Yaskawa INFORM job: pointsmerc3TRJ2.JBI

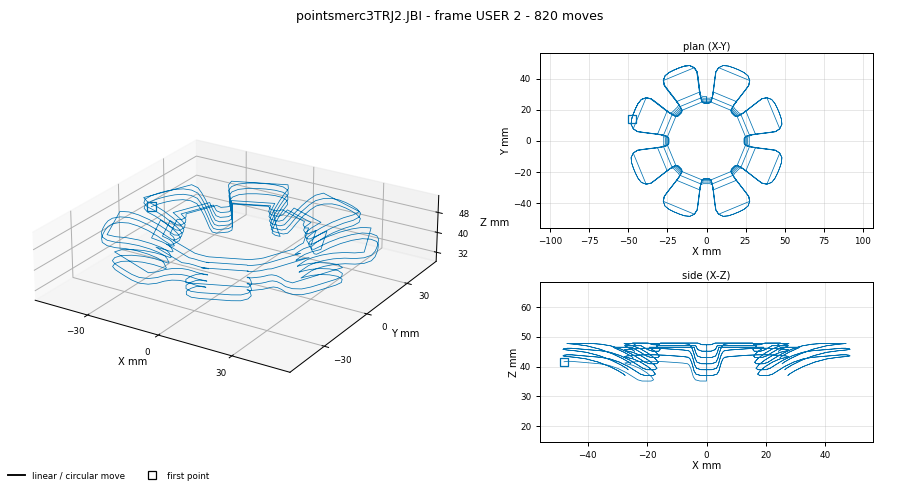
[picture p0: tool path of pointsmerc3TRJ2.JBI in frame USER 2, 820 of 820 moves have a stored position in this frame; points joined in program order, loops and branches not executed]
/JOB
//NAME pointsmerc3TRJ2
//POS
///NPOS 820,0,0,0,0,0
///USER 2
///TOOL 1
///POSTYPE USER
///RECTAN
///RCONF 1,0,0,0,0,0,0,0,0,0,0,0,0,0,0,0,0,0,0,0,0,0,0,0
C00000=-47.960,14.116,41.642,179.9713,-0.0983,0.0000
C00001=-46.852,17.458,41.781,179.9959,-0.0112,0.0000
C00002=-45.474,20.785,41.781,179.9950,-0.0108,0.0000
C00003=-43.894,23.932,41.642,179.9508,-0.0899,0.0000
C00004=-41.848,26.450,41.429,178.7336,-0.9130,0.0000
C00005=-38.982,27.526,41.216,176.7723,-0.3150,0.0000
C00006=-35.890,26.937,40.953,175.4165,2.2977,0.0000
C00007=-32.968,24.818,40.447,175.7483,3.1474,0.0000
C00008=-29.853,22.391,39.399,176.1159,2.8696,0.0000
C00009=-27.005,20.165,37.988,176.7172,2.3719,0.0000
C00010=-24.775,18.500,36.587,178.4223,1.0605,0.0000
C00011=-23.134,17.826,35.561,-161.2162,0.2646,0.0000
C00012=-21.719,18.610,35.152,-154.4517,19.2508,0.0000
C00013=-20.847,19.522,35.134,-156.6171,23.2444,0.0000
C00014=-20.193,20.193,35.146,-155.7569,22.3245,0.0000
C00015=-19.522,20.846,35.134,-154.9222,21.3860,0.0000
C00016=-18.610,21.719,35.152,-158.8420,24.0276,0.0000
C00017=-17.826,23.134,35.561,-179.7208,18.7831,0.0000
C00018=-18.500,24.775,36.587,-178.9391,-1.5774,0.0000
C00019=-20.165,27.005,37.988,-177.6242,-3.2800,0.0000
C00020=-22.391,29.853,39.399,-177.1238,-3.8792,0.0000
C00021=-24.818,32.968,40.447,-176.8439,-4.2453,0.0000
C00022=-26.937,35.890,40.953,-177.6949,-4.5798,0.0000
C00023=-27.526,38.982,41.216,179.6845,-3.2276,0.0000
C00024=-26.450,41.848,41.429,179.0868,-1.2662,0.0000
C00025=-23.932,43.894,41.642,179.9101,-0.0492,0.0000
C00026=-20.785,45.474,41.781,179.9892,-0.0050,0.0000
C00027=-17.458,46.852,41.781,179.9888,-0.0041,0.0000
C00028=-14.116,47.960,41.642,179.9017,-0.0287,0.0000
C00029=-10.888,48.294,41.429,178.4590,0.2497,0.0000
C00030=-8.101,47.028,41.216,177.4938,2.0588,0.0000
C00031=-6.331,44.425,40.953,178.3833,4.8651,0.0000
C00032=-5.763,40.861,40.447,179.2220,5.2308,0.0000
C00033=-5.276,36.942,39.399,179.2849,4.7747,0.0000
C00034=-4.837,33.354,37.988,179.3571,3.9980,0.0000
C00035=-4.437,30.601,36.587,179.6344,1.8654,0.0000
C00036=-3.753,28.963,35.561,-166.2914,-12.9686,0.0000
C00037=-2.199,28.517,35.152,-148.5463,-3.1419,0.0000
C00038=-0.937,28.545,35.134,-147.5179,1.2161,0.0000
C00039=0.000,28.557,35.146,-147.5083,-0.0008,0.0000
C00040=0.000,27.418,37.029,-150.2670,-0.0007,0.0000
C00041=0.833,27.409,37.016,-150.2716,-1.0327,0.0000
C00042=2.024,27.393,37.035,-151.4315,3.4006,0.0000
C00043=3.544,27.900,37.475,-168.9217,11.4487,0.0000
C00044=4.196,29.693,38.576,179.6272,-2.1342,0.0000
C00045=4.590,32.667,40.064,179.4709,-3.5322,0.0000
C00046=5.044,36.489,41.539,179.4511,-3.8692,0.0000
C00047=5.547,40.603,42.621,179.4411,-3.9829,0.0000
C00048=6.113,44.307,43.139,178.8534,-3.5959,0.0000
C00049=7.904,47.004,43.407,178.1982,-1.5163,0.0000
C00050=10.737,48.321,43.623,178.9014,-0.1851,0.0000
C00051=14.024,47.990,43.840,179.9308,0.0202,0.0000
C00052=17.428,46.864,43.981,179.9923,0.0029,0.0000
C00053=20.814,45.461,43.981,179.9925,0.0034,0.0000
C00054=24.018,43.851,43.840,179.9368,0.0347,0.0000
C00055=26.576,41.761,43.623,179.3540,0.9077,0.0000
C00056=27.648,38.826,43.407,179.7985,2.3462,0.0000
C00057=27.007,35.652,43.139,-178.2649,3.3521,0.0000
C00058=24.788,32.633,42.621,-177.5757,3.2100,0.0000
C00059=22.235,29.369,41.539,-177.6492,3.1226,0.0000
C00060=19.854,26.344,40.064,-177.8742,2.8707,0.0000
C00061=18.029,23.963,38.576,-178.7540,1.7725,0.0000
C00062=17.223,22.234,37.475,179.5719,-15.8740,0.0000
C00063=17.939,20.801,37.035,-161.3669,-22.3022,0.0000
C00064=18.793,19.970,37.016,-157.2922,-19.7457,0.0000
C00065=19.387,19.387,37.029,-158.0073,-20.5293,0.0000
C00066=19.970,18.793,37.016,-158.7389,-21.3057,0.0000
C00067=20.801,17.939,37.035,-156.5931,-17.1916,0.0000
C00068=22.234,17.223,37.475,-164.1263,0.4121,0.0000
C00069=23.963,18.029,38.576,178.2271,-1.2454,0.0000
C00070=26.344,19.854,40.064,177.1273,-2.1231,0.0000
C00071=29.369,22.235,41.539,176.8747,-2.3473,0.0000
C00072=32.633,24.788,42.621,176.7872,-2.4205,0.0000
C00073=35.652,27.007,43.139,176.6464,-1.7322,0.0000
C00074=38.826,27.648,43.407,177.6538,0.2014,0.0000
C00075=41.761,26.576,43.623,179.0922,0.6459,0.0000
C00076=43.851,24.018,43.840,179.9653,0.0632,0.0000
C00077=45.461,20.814,43.981,179.9966,0.0075,0.0000
C00078=46.864,17.428,43.981,179.9971,0.0077,0.0000
C00079=47.990,14.024,43.840,179.9798,0.0692,0.0000
C00080=48.321,10.737,43.623,-179.8148,1.0986,0.0000
C00081=47.004,7.904,43.407,-178.4829,1.8012,0.0000
C00082=44.307,6.113,43.139,-176.4033,1.1444,0.0000
C00083=40.603,5.547,42.621,-176.0170,0.5575,0.0000
C00084=36.489,5.044,41.539,-176.1306,0.5476,0.0000
C00085=32.667,4.590,40.064,-176.4677,0.5281,0.0000
C00086=29.693,4.196,38.576,-177.8658,0.3726,0.0000
C00087=27.900,3.544,37.475,168.3398,-10.8552,0.0000
C00088=27.393,2.024,37.035,176.1294,-28.5136,0.0000
C00089=27.409,0.833,37.016,-178.8108,-29.7231,0.0000
C00090=27.418,0.000,37.029,-179.9991,-29.7330,0.0000
C00091=27.409,-0.832,37.016,178.8099,-29.7231,0.0000
C00092=27.393,-2.024,37.035,-176.1268,-28.5126,0.0000
C00093=27.900,-3.544,37.475,-168.3400,-10.8545,0.0000
C00094=29.693,-4.196,38.576,177.8658,0.3726,0.0000
C00095=32.667,-4.590,40.064,176.4677,0.5281,0.0000
C00096=36.489,-5.044,41.539,176.1306,0.5476,0.0000
C00097=40.603,-5.547,42.621,176.0170,0.5575,0.0000
C00098=44.307,-6.113,43.139,176.4033,1.1444,0.0000
C00099=47.004,-7.904,43.407,178.4829,1.8012,0.0000
C00100=48.321,-10.737,43.623,179.8148,1.0986,0.0000
C00101=47.990,-14.024,43.840,-179.9798,0.0692,0.0000
C00102=46.864,-17.428,43.981,-179.9971,0.0077,0.0000
C00103=45.461,-20.814,43.981,-179.9966,0.0075,0.0000
C00104=43.851,-24.018,43.840,-179.9653,0.0632,0.0000
C00105=41.761,-26.576,43.623,-179.0922,0.6459,0.0000
C00106=38.826,-27.648,43.407,-177.6538,0.2014,0.0000
C00107=35.652,-27.007,43.139,-176.6464,-1.7322,0.0000
C00108=32.633,-24.788,42.621,-176.7872,-2.4205,0.0000
C00109=29.369,-22.235,41.539,-176.8747,-2.3473,0.0000
C00110=26.344,-19.854,40.064,-177.1273,-2.1231,0.0000
C00111=23.963,-18.029,38.576,-178.2271,-1.2454,0.0000
C00112=22.234,-17.223,37.475,164.1256,0.4118,0.0000
C00113=20.801,-17.939,37.035,156.5939,-17.1939,0.0000
C00114=19.970,-18.793,37.016,158.7383,-21.3051,0.0000
C00115=19.387,-19.387,37.029,158.0084,-20.5305,0.0000
C00116=18.793,-19.970,37.016,157.2916,-19.7451,0.0000
C00117=17.939,-20.801,37.035,161.3693,-22.3033,0.0000
C00118=17.223,-22.234,37.475,-179.5715,-15.8733,0.0000
C00119=18.029,-23.963,38.576,178.7540,1.7725,0.0000
C00120=19.854,-26.344,40.064,177.8742,2.8707,0.0000
C00121=22.235,-29.369,41.539,177.6492,3.1226,0.0000
C00122=24.788,-32.633,42.621,177.5757,3.2100,0.0000
C00123=27.007,-35.652,43.139,178.2649,3.3521,0.0000
C00124=27.648,-38.826,43.407,-179.7985,2.3462,0.0000
C00125=26.576,-41.761,43.623,-179.3540,0.9077,0.0000
C00126=24.018,-43.851,43.840,-179.9368,0.0347,0.0000
C00127=20.814,-45.461,43.981,-179.9925,0.0034,0.0000
C00128=17.428,-46.864,43.981,-179.9923,0.0029,0.0000
C00129=14.024,-47.990,43.840,-179.9308,0.0202,0.0000
C00130=10.737,-48.321,43.623,-178.9014,-0.1851,0.0000
C00131=7.904,-47.004,43.407,-178.1982,-1.5163,0.0000
C00132=6.113,-44.307,43.139,-178.8534,-3.5959,0.0000
C00133=5.547,-40.603,42.621,-179.4411,-3.9829,0.0000
C00134=5.044,-36.489,41.539,-179.4511,-3.8692,0.0000
C00135=4.590,-32.667,40.064,-179.4709,-3.5322,0.0000
C00136=4.196,-29.693,38.576,-179.6272,-2.1342,0.0000
C00137=3.544,-27.900,37.475,168.9217,11.4487,0.0000
C00138=2.024,-27.393,37.035,151.4315,3.4006,0.0000
C00139=0.833,-27.409,37.016,150.2716,-1.0327,0.0000
C00140=0.000,-27.418,37.029,150.2670,-0.0007,0.0000
C00141=0.000,-27.418,37.029,150.2670,-0.0007,0.0000
C00142=-0.832,-27.409,37.016,150.2716,1.0335,0.0000
C00143=-2.024,-27.393,37.035,151.4324,-3.4028,0.0000
C00144=-3.544,-27.900,37.475,168.9224,-11.4486,0.0000
C00145=-4.196,-29.693,38.576,-179.6272,2.1342,0.0000
C00146=-4.590,-32.667,40.064,-179.4709,3.5322,0.0000
C00147=-5.044,-36.489,41.539,-179.4511,3.8692,0.0000
C00148=-5.547,-40.603,42.621,-179.4411,3.9829,0.0000
C00149=-6.113,-44.307,43.139,-178.8534,3.5959,0.0000
C00150=-7.904,-47.004,43.407,-178.1982,1.5163,0.0000
C00151=-10.737,-48.321,43.623,-178.9014,0.1851,0.0000
C00152=-14.024,-47.990,43.840,-179.9308,-0.0202,0.0000
C00153=-17.428,-46.864,43.981,-179.9923,-0.0029,0.0000
C00154=-20.814,-45.461,43.981,-179.9925,-0.0034,0.0000
C00155=-24.018,-43.851,43.840,-179.9368,-0.0347,0.0000
C00156=-26.576,-41.761,43.623,-179.3540,-0.9077,0.0000
C00157=-27.648,-38.826,43.407,-179.7985,-2.3462,0.0000
C00158=-27.007,-35.652,43.139,178.2649,-3.3521,0.0000
C00159=-24.788,-32.633,42.621,177.5757,-3.2100,0.0000
C00160=-22.235,-29.369,41.539,177.6492,-3.1226,0.0000
C00161=-19.854,-26.344,40.064,177.8742,-2.8707,0.0000
C00162=-18.029,-23.963,38.576,178.7540,-1.7725,0.0000
C00163=-17.223,-22.234,37.475,-179.5719,15.8740,0.0000
C00164=-17.939,-20.801,37.035,161.3669,22.3022,0.0000
C00165=-18.793,-19.970,37.016,157.2922,19.7457,0.0000
C00166=-19.387,-19.387,37.029,158.0073,20.5293,0.0000
C00167=-19.970,-18.793,37.016,158.7389,21.3057,0.0000
C00168=-20.801,-17.939,37.035,156.5931,17.1916,0.0000
C00169=-22.234,-17.223,37.475,164.1263,-0.4121,0.0000
C00170=-23.963,-18.029,38.576,-178.2271,1.2454,0.0000
C00171=-26.344,-19.854,40.064,-177.1273,2.1231,0.0000
C00172=-29.369,-22.235,41.539,-176.8747,2.3473,0.0000
C00173=-32.633,-24.788,42.621,-176.7872,2.4205,0.0000
C00174=-35.652,-27.007,43.139,-176.6464,1.7322,0.0000
C00175=-38.826,-27.648,43.407,-177.6538,-0.2014,0.0000
C00176=-41.761,-26.576,43.623,-179.0922,-0.6459,0.0000
C00177=-43.851,-24.018,43.840,-179.9653,-0.0632,0.0000
C00178=-45.461,-20.814,43.981,-179.9966,-0.0075,0.0000
C00179=-46.864,-17.428,43.981,-179.9971,-0.0077,0.0000
C00180=-47.990,-14.024,43.840,-179.9798,-0.0692,0.0000
C00181=-48.321,-10.737,43.623,179.8148,-1.0986,0.0000
C00182=-47.004,-7.904,43.407,178.4829,-1.8012,0.0000
C00183=-44.307,-6.113,43.139,176.4033,-1.1444,0.0000
C00184=-40.603,-5.547,42.621,176.0170,-0.5575,0.0000
C00185=-36.489,-5.044,41.539,176.1306,-0.5476,0.0000
C00186=-32.667,-4.590,40.064,176.4677,-0.5281,0.0000
C00187=-29.693,-4.196,38.576,177.8658,-0.3726,0.0000
C00188=-27.900,-3.544,37.475,-168.3398,10.8552,0.0000
C00189=-27.393,-2.024,37.035,-176.1294,28.5136,0.0000
C00190=-27.409,-0.833,37.016,178.8108,29.7231,0.0000
C00191=-27.418,0.000,37.029,179.9991,29.7330,0.0000
C00192=-27.409,0.832,37.016,-178.8099,29.7231,0.0000
C00193=-27.393,2.024,37.035,176.1268,28.5126,0.0000
C00194=-27.900,3.544,37.475,168.3400,10.8545,0.0000
C00195=-29.693,4.196,38.576,-177.8658,-0.3726,0.0000
C00196=-32.667,4.590,40.064,-176.4677,-0.5281,0.0000
C00197=-36.489,5.044,41.539,-176.1306,-0.5476,0.0000
C00198=-40.603,5.547,42.621,-176.0170,-0.5575,0.0000
C00199=-44.307,6.113,43.139,-176.4033,-1.1444,0.0000
C00200=-47.004,7.904,43.407,-178.4829,-1.8012,0.0000
C00201=-48.321,10.737,43.623,-179.8148,-1.0986,0.0000
C00202=-47.990,14.024,43.840,179.9798,-0.0692,0.0000
C00203=-46.864,17.428,43.981,179.9971,-0.0077,0.0000
C00204=-45.461,20.814,43.981,179.9966,-0.0075,0.0000
C00205=-43.851,24.018,43.840,179.9653,-0.0632,0.0000
C00206=-41.761,26.576,43.623,179.0922,-0.6459,0.0000
C00207=-38.826,27.648,43.407,177.6538,-0.2014,0.0000
C00208=-35.652,27.007,43.139,176.6464,1.7322,0.0000
C00209=-32.633,24.788,42.621,176.7872,2.4205,0.0000
C00210=-29.369,22.235,41.539,176.8747,2.3473,0.0000
C00211=-26.344,19.854,40.064,177.1273,2.1231,0.0000
C00212=-23.963,18.029,38.576,178.2271,1.2454,0.0000
C00213=-22.234,17.223,37.475,-164.1256,-0.4118,0.0000
C00214=-20.801,17.939,37.035,-156.5939,17.1939,0.0000
C00215=-19.970,18.793,37.016,-158.7383,21.3051,0.0000
C00216=-19.387,19.387,37.029,-158.0084,20.5305,0.0000
C00217=-18.793,19.970,37.016,-157.2916,19.7451,0.0000
C00218=-17.939,20.801,37.035,-161.3693,22.3033,0.0000
C00219=-17.223,22.234,37.475,179.5715,15.8733,0.0000
C00220=-18.029,23.963,38.576,-178.7540,-1.7725,0.0000
C00221=-19.854,26.344,40.064,-177.8742,-2.8707,0.0000
C00222=-22.235,29.369,41.539,-177.6492,-3.1226,0.0000
C00223=-24.788,32.633,42.621,-177.5757,-3.2100,0.0000
C00224=-27.007,35.652,43.139,-178.2649,-3.3521,0.0000
C00225=-27.648,38.826,43.407,179.7985,-2.3462,0.0000
C00226=-26.576,41.761,43.623,179.3540,-0.9077,0.0000
C00227=-24.018,43.851,43.840,179.9368,-0.0347,0.0000
C00228=-20.814,45.461,43.981,179.9925,-0.0034,0.0000
C00229=-17.428,46.864,43.981,179.9923,-0.0029,0.0000
C00230=-14.024,47.990,43.840,179.9308,-0.0202,0.0000
C00231=-10.737,48.321,43.623,178.9014,0.1851,0.0000
C00232=-7.904,47.004,43.407,178.1982,1.5163,0.0000
C00233=-6.113,44.307,43.139,178.8534,3.5959,0.0000
C00234=-5.547,40.603,42.621,179.4411,3.9829,0.0000
C00235=-5.044,36.489,41.539,179.4511,3.8692,0.0000
C00236=-4.590,32.667,40.064,179.4709,3.5322,0.0000
C00237=-4.196,29.693,38.576,179.6272,2.1342,0.0000
C00238=-3.544,27.900,37.475,-168.9224,-11.4486,0.0000
C00239=-2.024,27.393,37.035,-151.4324,-3.4028,0.0000
C00240=-0.832,27.409,37.016,-150.2716,1.0335,0.0000
C00241=0.000,27.418,37.029,-150.2670,-0.0007,0.0000
C00242=0.000,26.383,38.970,-153.7508,-0.0006,0.0000
C00243=0.738,26.377,38.956,-153.7490,-0.8316,0.0000
C00244=1.865,26.371,38.977,-154.9962,3.4534,0.0000
C00245=3.355,26.945,39.448,-171.3719,9.6260,0.0000
C00246=3.987,28.902,40.618,179.6696,-2.0938,0.0000
C00247=4.387,32.102,42.180,179.5989,-2.8366,0.0000
C00248=4.868,36.145,43.705,179.6256,-2.7489,0.0000
C00249=5.395,40.422,44.808,179.6621,-2.5077,0.0000
C00250=5.967,44.227,45.333,179.3497,-2.0954,0.0000
C00251=7.777,46.989,45.603,179.0076,-0.8478,0.0000
C00252=10.643,48.338,45.821,179.4199,-0.1001,0.0000
C00253=13.968,48.009,46.039,179.9653,0.0101,0.0000
C00254=17.410,46.871,46.181,179.9963,0.0014,0.0000
C00255=20.832,45.453,46.181,179.9964,0.0017,0.0000
C00256=24.070,43.824,46.039,179.9683,0.0174,0.0000
C00257=26.655,41.706,45.821,179.6606,0.4809,0.0000
C00258=27.727,38.725,45.603,179.8978,1.3012,0.0000
C00259=27.054,35.493,45.333,-178.9775,1.9413,0.0000
C00260=24.768,32.397,44.808,-178.4649,2.0118,0.0000
C00261=22.116,29.001,43.705,-178.3199,2.2080,0.0000
C00262=19.598,25.801,42.180,-178.2767,2.2889,0.0000
C00263=17.618,23.256,40.618,-178.7526,1.7139,0.0000
C00264=16.680,21.426,39.448,179.1975,-12.8751,0.0000
C00265=17.329,19.966,38.977,-164.2142,-19.9336,0.0000
C00266=18.130,19.173,38.956,-160.1927,-17.6055,0.0000
C00267=18.656,18.656,38.970,-160.7762,-18.2238,0.0000
C00268=19.173,18.130,38.956,-161.3623,-18.8441,0.0000
C00269=19.966,17.329,38.977,-159.3493,-14.8154,0.0000
C00270=21.426,16.680,39.448,-167.1244,0.7826,0.0000
C00271=23.256,17.618,40.618,178.2857,-1.2468,0.0000
C00272=25.801,19.598,42.180,177.7101,-1.7220,0.0000
C00273=29.001,22.116,43.705,177.7910,-1.6789,0.0000
C00274=32.397,24.768,44.808,177.9875,-1.5342,0.0000
C00275=35.493,27.054,45.333,178.0584,-1.0219,0.0000
C00276=38.725,27.727,45.603,178.6988,0.1021,0.0000
C00277=41.706,26.655,45.821,179.5191,0.3394,0.0000
C00278=43.824,24.070,46.039,179.9826,0.0317,0.0000
C00279=45.453,20.832,46.181,179.9983,0.0036,0.0000
C00280=46.871,17.410,46.181,179.9986,0.0037,0.0000
C00281=48.009,13.968,46.039,179.9899,0.0347,0.0000
C00282=48.338,10.643,45.821,-179.8999,0.5801,0.0000
C00283=46.989,7.777,45.603,-179.1520,0.9923,0.0000
C00284=44.227,5.967,45.333,-177.9044,0.6499,0.0000
C00285=40.422,5.395,44.808,-177.4922,0.3376,0.0000
C00286=36.145,4.868,43.705,-177.2510,0.3740,0.0000
C00287=32.102,4.387,42.180,-177.1633,0.4006,0.0000
C00288=28.902,3.987,40.618,-177.9062,0.3302,0.0000
C00289=26.945,3.355,39.448,170.2659,-8.5057,0.0000
C00290=26.371,1.865,38.977,176.1905,-24.9553,0.0000
C00291=26.377,0.738,38.956,-179.0728,-26.2481,0.0000
C00292=26.383,0.000,38.970,-179.9993,-26.2492,0.0000
C00293=26.377,-0.738,38.956,179.0721,-26.2481,0.0000
C00294=26.371,-1.865,38.977,-176.1882,-24.9543,0.0000
C00295=26.945,-3.355,39.448,-170.2662,-8.5050,0.0000
C00296=28.902,-3.987,40.618,177.9062,0.3302,0.0000
C00297=32.102,-4.387,42.180,177.1633,0.4006,0.0000
C00298=36.145,-4.868,43.705,177.2510,0.3740,0.0000
C00299=40.422,-5.395,44.808,177.4922,0.3376,0.0000
C00300=44.227,-5.967,45.333,177.9044,0.6499,0.0000
C00301=46.989,-7.777,45.603,179.1520,0.9923,0.0000
C00302=48.338,-10.643,45.821,179.8999,0.5801,0.0000
C00303=48.009,-13.968,46.039,-179.9899,0.0347,0.0000
C00304=46.871,-17.410,46.181,-179.9986,0.0037,0.0000
C00305=45.453,-20.832,46.181,-179.9983,0.0036,0.0000
C00306=43.824,-24.070,46.039,-179.9826,0.0317,0.0000
C00307=41.706,-26.655,45.821,-179.5191,0.3394,0.0000
C00308=38.725,-27.727,45.603,-178.6988,0.1021,0.0000
C00309=35.493,-27.054,45.333,-178.0584,-1.0219,0.0000
C00310=32.397,-24.768,44.808,-177.9875,-1.5342,0.0000
C00311=29.001,-22.116,43.705,-177.7910,-1.6789,0.0000
C00312=25.801,-19.598,42.180,-177.7101,-1.7220,0.0000
C00313=23.256,-17.618,40.618,-178.2857,-1.2468,0.0000
C00314=21.426,-16.680,39.448,167.1236,0.7823,0.0000
C00315=19.966,-17.329,38.977,159.3500,-14.8176,0.0000
C00316=19.173,-18.130,38.956,161.3618,-18.8436,0.0000
C00317=18.656,-18.656,38.970,160.7770,-18.2247,0.0000
C00318=18.130,-19.173,38.956,160.1923,-17.6051,0.0000
C00319=17.329,-19.966,38.977,164.2165,-19.9345,0.0000
C00320=16.680,-21.426,39.448,-179.1972,-12.8744,0.0000
C00321=17.618,-23.256,40.618,178.7526,1.7139,0.0000
C00322=19.598,-25.801,42.180,178.2767,2.2889,0.0000
C00323=22.116,-29.001,43.705,178.3199,2.2080,0.0000
C00324=24.768,-32.397,44.808,178.4649,2.0118,0.0000
C00325=27.054,-35.493,45.333,178.9775,1.9413,0.0000
C00326=27.727,-38.725,45.603,-179.8978,1.3012,0.0000
C00327=26.655,-41.706,45.821,-179.6606,0.4809,0.0000
C00328=24.070,-43.824,46.039,-179.9683,0.0174,0.0000
C00329=20.832,-45.453,46.181,-179.9964,0.0017,0.0000
C00330=17.410,-46.871,46.181,-179.9963,0.0014,0.0000
C00331=13.968,-48.009,46.039,-179.9653,0.0101,0.0000
C00332=10.643,-48.338,45.821,-179.4199,-0.1001,0.0000
C00333=7.777,-46.989,45.603,-179.0076,-0.8478,0.0000
C00334=5.967,-44.227,45.333,-179.3497,-2.0954,0.0000
C00335=5.395,-40.422,44.808,-179.6621,-2.5077,0.0000
C00336=4.868,-36.145,43.705,-179.6256,-2.7489,0.0000
C00337=4.387,-32.102,42.180,-179.5989,-2.8366,0.0000
C00338=3.987,-28.902,40.618,-179.6696,-2.0938,0.0000
C00339=3.355,-26.945,39.448,171.3719,9.6260,0.0000
C00340=1.865,-26.371,38.977,154.9962,3.4534,0.0000
C00341=0.738,-26.377,38.956,153.7490,-0.8316,0.0000
C00342=0.000,-26.383,38.970,153.7508,-0.0006,0.0000
C00343=0.000,-26.383,38.970,153.7508,-0.0006,0.0000
C00344=-0.738,-26.377,38.956,153.7490,0.8322,0.0000
C00345=-1.865,-26.371,38.977,154.9971,-3.4555,0.0000
C00346=-3.355,-26.945,39.448,171.3727,-9.6258,0.0000
C00347=-3.987,-28.902,40.618,-179.6696,2.0938,0.0000
C00348=-4.387,-32.102,42.180,-179.5989,2.8366,0.0000
C00349=-4.868,-36.145,43.705,-179.6256,2.7489,0.0000
C00350=-5.395,-40.422,44.808,-179.6621,2.5077,0.0000
C00351=-5.967,-44.227,45.333,-179.3497,2.0954,0.0000
C00352=-7.777,-46.989,45.603,-179.0076,0.8478,0.0000
C00353=-10.643,-48.338,45.821,-179.4199,0.1001,0.0000
C00354=-13.968,-48.009,46.039,-179.9653,-0.0101,0.0000
C00355=-17.410,-46.871,46.181,-179.9963,-0.0014,0.0000
C00356=-20.832,-45.453,46.181,-179.9964,-0.0017,0.0000
C00357=-24.070,-43.824,46.039,-179.9683,-0.0174,0.0000
C00358=-26.655,-41.706,45.821,-179.6606,-0.4809,0.0000
C00359=-27.727,-38.725,45.603,-179.8978,-1.3012,0.0000
C00360=-27.054,-35.493,45.333,178.9775,-1.9413,0.0000
C00361=-24.768,-32.397,44.808,178.4649,-2.0118,0.0000
C00362=-22.116,-29.001,43.705,178.3199,-2.2080,0.0000
C00363=-19.598,-25.801,42.180,178.2767,-2.2889,0.0000
C00364=-17.618,-23.256,40.618,178.7526,-1.7139,0.0000
C00365=-16.680,-21.426,39.448,-179.1975,12.8751,0.0000
C00366=-17.329,-19.966,38.977,164.2142,19.9336,0.0000
C00367=-18.130,-19.173,38.956,160.1927,17.6055,0.0000
C00368=-18.656,-18.656,38.970,160.7762,18.2238,0.0000
C00369=-19.173,-18.130,38.956,161.3623,18.8441,0.0000
C00370=-19.966,-17.329,38.977,159.3493,14.8154,0.0000
C00371=-21.426,-16.680,39.448,167.1244,-0.7826,0.0000
C00372=-23.256,-17.618,40.618,-178.2857,1.2468,0.0000
C00373=-25.801,-19.598,42.180,-177.7101,1.7220,0.0000
C00374=-29.001,-22.116,43.705,-177.7910,1.6789,0.0000
C00375=-32.397,-24.768,44.808,-177.9875,1.5342,0.0000
C00376=-35.493,-27.054,45.333,-178.0584,1.0219,0.0000
C00377=-38.725,-27.727,45.603,-178.6988,-0.1021,0.0000
C00378=-41.706,-26.655,45.821,-179.5191,-0.3394,0.0000
C00379=-43.824,-24.070,46.039,-179.9826,-0.0317,0.0000
C00380=-45.453,-20.832,46.181,-179.9983,-0.0036,0.0000
C00381=-46.871,-17.410,46.181,-179.9986,-0.0037,0.0000
C00382=-48.009,-13.968,46.039,-179.9899,-0.0347,0.0000
C00383=-48.338,-10.643,45.821,179.8999,-0.5801,0.0000
C00384=-46.989,-7.777,45.603,179.1520,-0.9923,0.0000
C00385=-44.227,-5.967,45.333,177.9044,-0.6499,0.0000
C00386=-40.422,-5.395,44.808,177.4922,-0.3376,0.0000
C00387=-36.145,-4.868,43.705,177.2510,-0.3740,0.0000
C00388=-32.102,-4.387,42.180,177.1633,-0.4006,0.0000
C00389=-28.902,-3.987,40.618,177.9062,-0.3302,0.0000
C00390=-26.945,-3.355,39.448,-170.2659,8.5057,0.0000
C00391=-26.371,-1.865,38.977,-176.1905,24.9553,0.0000
C00392=-26.377,-0.738,38.956,179.0728,26.2481,0.0000
C00393=-26.383,0.000,38.970,179.9993,26.2492,0.0000
C00394=-26.377,0.738,38.956,-179.0721,26.2481,0.0000
C00395=-26.371,1.865,38.977,176.1882,24.9543,0.0000
C00396=-26.945,3.355,39.448,170.2662,8.5050,0.0000
C00397=-28.902,3.987,40.618,-177.9062,-0.3302,0.0000
C00398=-32.102,4.387,42.180,-177.1633,-0.4006,0.0000
C00399=-36.145,4.868,43.705,-177.2510,-0.3740,0.0000
C00400=-40.422,5.395,44.808,-177.4922,-0.3376,0.0000
C00401=-44.227,5.967,45.333,-177.9044,-0.6499,0.0000
C00402=-46.989,7.777,45.603,-179.1520,-0.9923,0.0000
C00403=-48.338,10.643,45.821,-179.8999,-0.5801,0.0000
C00404=-48.009,13.968,46.039,179.9899,-0.0347,0.0000
C00405=-46.871,17.410,46.181,179.9986,-0.0037,0.0000
C00406=-45.453,20.832,46.181,179.9983,-0.0036,0.0000
C00407=-43.824,24.070,46.039,179.9826,-0.0317,0.0000
C00408=-41.706,26.655,45.821,179.5191,-0.3394,0.0000
C00409=-38.725,27.727,45.603,178.6988,-0.1021,0.0000
C00410=-35.493,27.054,45.333,178.0584,1.0219,0.0000
C00411=-32.397,24.768,44.808,177.9875,1.5342,0.0000
C00412=-29.001,22.116,43.705,177.7910,1.6789,0.0000
C00413=-25.801,19.598,42.180,177.7101,1.7220,0.0000
C00414=-23.256,17.618,40.618,178.2857,1.2468,0.0000
C00415=-21.426,16.680,39.448,-167.1236,-0.7823,0.0000
C00416=-19.966,17.329,38.977,-159.3500,14.8176,0.0000
C00417=-19.173,18.130,38.956,-161.3618,18.8436,0.0000
C00418=-18.656,18.656,38.970,-160.7770,18.2247,0.0000
C00419=-18.130,19.173,38.956,-160.1923,17.6051,0.0000
C00420=-17.329,19.966,38.977,-164.2165,19.9345,0.0000
C00421=-16.680,21.426,39.448,179.1972,12.8744,0.0000
C00422=-17.618,23.256,40.618,-178.7526,-1.7139,0.0000
C00423=-19.598,25.801,42.180,-178.2767,-2.2889,0.0000
C00424=-22.116,29.001,43.705,-178.3199,-2.2080,0.0000
C00425=-24.768,32.397,44.808,-178.4649,-2.0118,0.0000
C00426=-27.054,35.493,45.333,-178.9775,-1.9413,0.0000
C00427=-27.727,38.725,45.603,179.8978,-1.3012,0.0000
C00428=-26.655,41.706,45.821,179.6606,-0.4809,0.0000
C00429=-24.070,43.824,46.039,179.9683,-0.0174,0.0000
C00430=-20.832,45.453,46.181,179.9964,-0.0017,0.0000
C00431=-17.410,46.871,46.181,179.9963,-0.0014,0.0000
C00432=-13.968,48.009,46.039,179.9653,-0.0101,0.0000
C00433=-10.643,48.338,45.821,179.4199,0.1001,0.0000
C00434=-7.777,46.989,45.603,179.0076,0.8478,0.0000
C00435=-5.967,44.227,45.333,179.3497,2.0954,0.0000
C00436=-5.395,40.422,44.808,179.6621,2.5077,0.0000
C00437=-4.868,36.145,43.705,179.6256,2.7489,0.0000
C00438=-4.387,32.102,42.180,179.5989,2.8366,0.0000
C00439=-3.987,28.902,40.618,179.6696,2.0938,0.0000
C00440=-3.355,26.945,39.448,-171.3727,-9.6258,0.0000
C00441=-1.865,26.371,38.977,-154.9971,-3.4555,0.0000
C00442=-0.738,26.377,38.956,-153.7490,0.8322,0.0000
C00443=0.000,26.383,38.970,-153.7508,-0.0006,0.0000
C00444=0.000,25.483,40.978,-158.1137,-0.0004,0.0000
C00445=0.656,25.479,40.963,-158.1034,-0.6202,0.0000
C00446=1.726,25.483,40.985,-159.3485,3.2259,0.0000
C00447=3.194,26.129,41.485,-173.6456,7.5533,0.0000
C00448=3.816,28.261,42.716,179.7442,-1.7639,0.0000
C00449=4.237,31.687,44.335,179.7389,-1.9261,0.0000
C00450=4.757,35.929,45.891,179.8102,-1.4294,0.0000
C00451=5.317,40.329,47.005,179.8913,-0.8234,0.0000
C00452=5.904,44.193,47.531,179.8811,-0.3876,0.0000
C00453=7.727,46.983,47.803,179.9143,-0.0736,0.0000
C00454=27.758,38.686,47.803,179.9915,0.1126,0.0000
C00455=27.074,35.424,47.531,-179.8100,0.3581,0.0000
C00456=24.758,32.277,47.005,-179.4946,0.6591,0.0000
C00457=22.041,28.769,45.891,-179.1233,1.1448,0.0000
C00458=19.410,25.402,44.335,-178.8223,1.5464,0.0000
C00459=17.285,22.682,42.716,-178.9333,1.4280,0.0000
C00460=16.217,20.734,41.485,179.1065,-9.8187,0.0000
C00461=16.798,19.240,40.985,-167.3786,-16.7849,0.0000
C00462=17.553,18.480,40.963,-163.6981,-14.8348,0.0000
C00463=18.019,18.019,40.978,-164.1420,-15.2826,0.0000
C00464=18.480,17.553,40.963,-164.5731,-15.7444,0.0000
C00465=19.240,16.798,40.985,-162.8231,-12.0734,0.0000
C00466=20.735,16.217,41.485,-170.1809,0.8807,0.0000
C00467=22.682,17.285,42.716,178.5717,-1.0663,0.0000
C00468=25.402,19.410,44.335,178.4533,-1.1773,0.0000
C00469=28.769,22.041,45.891,178.8550,-0.8765,0.0000
C00470=32.277,24.758,47.005,179.3409,-0.5054,0.0000
C00471=35.424,27.074,47.531,179.6419,-0.1900,0.0000
C00472=38.686,27.758,47.803,179.8874,0.0085,0.0000
C00473=46.983,7.727,47.803,-179.9264,0.0857,0.0000
C00474=44.193,5.904,47.531,-179.6124,0.1189,0.0000
C00475=40.329,5.317,47.005,-179.1766,0.1086,0.0000
C00476=35.929,4.757,45.891,-178.5706,0.1897,0.0000
C00477=31.687,4.237,44.335,-178.0739,0.2609,0.0000
C00478=28.261,3.816,42.716,-178.2360,0.2557,0.0000
C00479=26.129,3.194,41.485,172.4006,-6.2991,0.0000
C00480=25.483,1.726,40.985,176.5531,-20.6173,0.0000
C00481=25.479,0.656,40.963,-179.3316,-21.8952,0.0000
C00482=25.483,0.000,40.978,-179.9995,-21.8863,0.0000
C00483=25.479,-0.655,40.963,179.3311,-21.8952,0.0000
C00484=25.483,-1.727,40.985,-176.5512,-20.6163,0.0000
C00485=26.129,-3.194,41.485,-172.4009,-6.2984,0.0000
C00486=28.261,-3.816,42.716,178.2360,0.2557,0.0000
C00487=31.687,-4.237,44.335,178.0739,0.2609,0.0000
C00488=35.929,-4.757,45.891,178.5706,0.1897,0.0000
C00489=40.329,-5.317,47.005,179.1766,0.1086,0.0000
C00490=44.193,-5.904,47.531,179.6124,0.1189,0.0000
C00491=46.983,-7.727,47.803,179.9264,0.0857,0.0000
C00492=38.686,-27.758,47.803,-179.8874,0.0085,0.0000
C00493=35.424,-27.074,47.531,-179.6419,-0.1900,0.0000
C00494=32.277,-24.758,47.005,-179.3409,-0.5054,0.0000
C00495=28.769,-22.041,45.891,-178.8550,-0.8765,0.0000
C00496=25.402,-19.410,44.335,-178.4533,-1.1773,0.0000
C00497=22.682,-17.285,42.716,-178.5717,-1.0663,0.0000
C00498=20.734,-16.217,41.485,170.1802,0.8804,0.0000
C00499=19.240,-16.798,40.985,162.8237,-12.0754,0.0000
C00500=18.480,-17.553,40.963,164.5728,-15.7441,0.0000
C00501=18.019,-18.019,40.978,164.1426,-15.2833,0.0000
C00502=17.553,-18.480,40.963,163.6979,-14.8345,0.0000
C00503=16.798,-19.240,40.985,167.3807,-16.7856,0.0000
C00504=16.217,-20.735,41.485,-179.1062,-9.8180,0.0000
C00505=17.285,-22.682,42.716,178.9333,1.4280,0.0000
C00506=19.410,-25.402,44.335,178.8223,1.5464,0.0000
C00507=22.041,-28.769,45.891,179.1233,1.1448,0.0000
C00508=24.758,-32.277,47.005,179.4946,0.6591,0.0000
C00509=27.074,-35.424,47.531,179.8100,0.3581,0.0000
C00510=27.758,-38.686,47.803,-179.9915,0.1126,0.0000
C00511=7.727,-46.983,47.803,-179.9143,-0.0736,0.0000
C00512=5.904,-44.193,47.531,-179.8811,-0.3876,0.0000
C00513=5.317,-40.329,47.005,-179.8913,-0.8234,0.0000
C00514=4.757,-35.929,45.891,-179.8102,-1.4294,0.0000
C00515=4.237,-31.687,44.335,-179.7389,-1.9261,0.0000
C00516=3.816,-28.261,42.716,-179.7442,-1.7639,0.0000
C00517=3.194,-26.129,41.485,173.6456,7.5533,0.0000
C00518=1.726,-25.483,40.985,159.3485,3.2259,0.0000
C00519=0.656,-25.479,40.963,158.1034,-0.6202,0.0000
C00520=0.000,-25.483,40.978,158.1137,-0.0004,0.0000
C00521=0.000,-25.483,40.978,158.1137,-0.0004,0.0000
C00522=-0.655,-25.479,40.963,158.1034,0.6206,0.0000
C00523=-1.727,-25.483,40.985,159.3495,-3.2277,0.0000
C00524=-3.194,-26.129,41.485,173.6463,-7.5530,0.0000
C00525=-3.816,-28.261,42.716,-179.7442,1.7639,0.0000
C00526=-4.237,-31.687,44.335,-179.7389,1.9261,0.0000
C00527=-4.757,-35.929,45.891,-179.8102,1.4294,0.0000
C00528=-5.317,-40.329,47.005,-179.8913,0.8234,0.0000
C00529=-5.904,-44.193,47.531,-179.8811,0.3876,0.0000
C00530=-7.727,-46.983,47.803,-179.9143,0.0736,0.0000
C00531=-27.758,-38.686,47.803,-179.9915,-0.1126,0.0000
C00532=-27.074,-35.424,47.531,179.8100,-0.3581,0.0000
C00533=-24.758,-32.277,47.005,179.4946,-0.6591,0.0000
C00534=-22.041,-28.769,45.891,179.1233,-1.1448,0.0000
C00535=-19.410,-25.402,44.335,178.8223,-1.5464,0.0000
C00536=-17.285,-22.682,42.716,178.9333,-1.4280,0.0000
C00537=-16.217,-20.734,41.485,-179.1065,9.8187,0.0000
C00538=-16.798,-19.240,40.985,167.3786,16.7849,0.0000
C00539=-17.553,-18.480,40.963,163.6981,14.8348,0.0000
C00540=-18.019,-18.019,40.978,164.1420,15.2826,0.0000
C00541=-18.480,-17.553,40.963,164.5731,15.7444,0.0000
C00542=-19.240,-16.798,40.985,162.8231,12.0734,0.0000
C00543=-20.735,-16.217,41.485,170.1809,-0.8807,0.0000
C00544=-22.682,-17.285,42.716,-178.5717,1.0663,0.0000
C00545=-25.402,-19.410,44.335,-178.4533,1.1773,0.0000
C00546=-28.769,-22.041,45.891,-178.8550,0.8765,0.0000
C00547=-32.277,-24.758,47.005,-179.3409,0.5054,0.0000
C00548=-35.424,-27.074,47.531,-179.6419,0.1900,0.0000
C00549=-38.686,-27.758,47.803,-179.8874,-0.0085,0.0000
C00550=-46.983,-7.727,47.803,179.9264,-0.0857,0.0000
C00551=-44.193,-5.904,47.531,179.6124,-0.1189,0.0000
C00552=-40.329,-5.317,47.005,179.1766,-0.1086,0.0000
C00553=-35.929,-4.757,45.891,178.5706,-0.1897,0.0000
C00554=-31.687,-4.237,44.335,178.0739,-0.2609,0.0000
C00555=-28.261,-3.816,42.716,178.2360,-0.2557,0.0000
C00556=-26.129,-3.194,41.485,-172.4006,6.2991,0.0000
C00557=-25.483,-1.726,40.985,-176.5531,20.6173,0.0000
C00558=-25.479,-0.656,40.963,179.3316,21.8952,0.0000
C00559=-25.483,0.000,40.978,179.9995,21.8863,0.0000
C00560=-25.479,0.655,40.963,-179.3311,21.8952,0.0000
C00561=-25.483,1.727,40.985,176.5512,20.6163,0.0000
C00562=-26.129,3.194,41.485,172.4009,6.2984,0.0000
C00563=-28.261,3.816,42.716,-178.2360,-0.2557,0.0000
C00564=-31.687,4.237,44.335,-178.0739,-0.2609,0.0000
C00565=-35.929,4.757,45.891,-178.5706,-0.1897,0.0000
C00566=-40.329,5.317,47.005,-179.1766,-0.1086,0.0000
C00567=-44.193,5.904,47.531,-179.6124,-0.1189,0.0000
C00568=-46.983,7.727,47.803,-179.9264,-0.0857,0.0000
C00569=-38.686,27.758,47.803,179.8874,-0.0085,0.0000
C00570=-35.424,27.074,47.531,179.6419,0.1900,0.0000
C00571=-32.277,24.758,47.005,179.3409,0.5054,0.0000
C00572=-28.769,22.041,45.891,178.8550,0.8765,0.0000
C00573=-25.402,19.410,44.335,178.4533,1.1773,0.0000
C00574=-22.682,17.285,42.716,178.5717,1.0663,0.0000
C00575=-20.734,16.217,41.485,-170.1802,-0.8804,0.0000
C00576=-19.240,16.798,40.985,-162.8237,12.0754,0.0000
C00577=-18.480,17.553,40.963,-164.5728,15.7441,0.0000
C00578=-18.019,18.019,40.978,-164.1426,15.2833,0.0000
C00579=-17.553,18.480,40.963,-163.6979,14.8345,0.0000
C00580=-16.798,19.240,40.985,-167.3807,16.7856,0.0000
C00581=-16.217,20.735,41.485,179.1062,9.8180,0.0000
C00582=-17.285,22.682,42.716,-178.9333,-1.4280,0.0000
C00583=-19.410,25.402,44.335,-178.8223,-1.5464,0.0000
C00584=-22.041,28.769,45.891,-179.1233,-1.1448,0.0000
C00585=-24.758,32.277,47.005,-179.4946,-0.6591,0.0000
C00586=-27.074,35.424,47.531,-179.8100,-0.3581,0.0000
C00587=-27.758,38.686,47.803,179.9915,-0.1126,0.0000
C00588=-7.727,46.983,47.803,179.9143,0.0736,0.0000
C00589=-5.904,44.193,47.531,179.8811,0.3876,0.0000
C00590=-5.317,40.329,47.005,179.8913,0.8234,0.0000
C00591=-4.757,35.929,45.891,179.8102,1.4294,0.0000
C00592=-4.237,31.687,44.335,179.7389,1.9261,0.0000
C00593=-3.816,28.261,42.716,179.7442,1.7639,0.0000
C00594=-3.194,26.129,41.485,-173.6463,-7.5530,0.0000
C00595=-1.727,25.483,40.985,-159.3495,-3.2277,0.0000
C00596=-0.655,25.479,40.963,-158.1034,0.6206,0.0000
C00597=0.000,25.483,40.978,-158.1137,-0.0004,0.0000
C00598=0.000,24.757,43.054,-163.5138,-0.0002,0.0000
C00599=0.589,24.754,43.039,-163.4920,-0.4122,0.0000
C00600=1.615,24.766,43.062,-164.5921,2.6504,0.0000
C00601=3.068,25.489,43.586,-175.7793,5.2659,0.0000
C00602=3.695,27.804,44.865,179.8395,-1.1765,0.0000
C00603=4.151,31.448,46.521,179.8907,-0.8261,0.0000
C00604=19.301,25.172,46.521,-179.4931,0.6614,0.0000
C00605=17.048,22.273,44.865,-179.2815,0.9454,0.0000
C00606=15.854,20.193,43.586,179.2457,-6.7028,0.0000
C00607=16.370,18.654,43.062,-170.8582,-12.7306,0.0000
C00608=17.087,17.920,43.039,-167.8734,-11.2933,0.0000
C00609=17.506,17.506,43.054,-168.1802,-11.5757,0.0000
C00610=17.920,17.087,43.039,-168.4559,-11.8884,0.0000
C00611=18.654,16.370,43.062,-167.1106,-8.9135,0.0000
C00612=20.193,15.854,43.586,-173.2972,0.7493,0.0000
C00613=22.273,17.048,44.865,179.0546,-0.7184,0.0000
C00614=25.172,19.301,46.521,179.3386,-0.5068,0.0000
C00615=31.448,4.151,46.521,-179.1739,0.1093,0.0000
C00616=27.804,3.695,44.865,-178.8235,0.1604,0.0000
C00617=25.489,3.068,43.586,174.7199,-4.2029,0.0000
C00618=24.766,1.615,43.062,177.2510,-15.3911,0.0000
C00619=24.754,0.589,43.039,-179.5701,-16.5075,0.0000
C00620=24.757,0.000,43.054,-179.9998,-16.4862,0.0000
C00621=24.754,-0.589,43.039,179.5700,-16.5075,0.0000
C00622=24.766,-1.615,43.062,-177.2494,-15.3902,0.0000
C00623=25.489,-3.068,43.586,-174.7201,-4.2024,0.0000
C00624=27.804,-3.695,44.865,178.8235,0.1604,0.0000
C00625=31.448,-4.151,46.521,179.1739,0.1093,0.0000
C00626=25.172,-19.301,46.521,-179.3386,-0.5068,0.0000
C00627=22.273,-17.048,44.865,-179.0546,-0.7184,0.0000
C00628=20.193,-15.854,43.586,173.2966,0.7491,0.0000
C00629=18.654,-16.370,43.062,167.1110,-8.9152,0.0000
C00630=17.920,-17.087,43.039,168.4558,-11.8883,0.0000
C00631=17.506,-17.506,43.054,168.1805,-11.5761,0.0000
C00632=17.087,-17.920,43.039,167.8733,-11.2932,0.0000
C00633=16.370,-18.654,43.062,170.8599,-12.7311,0.0000
C00634=15.854,-20.193,43.586,-179.2456,-6.7022,0.0000
C00635=17.048,-22.273,44.865,179.2815,0.9454,0.0000
C00636=19.301,-25.172,46.521,179.4931,0.6614,0.0000
C00637=4.151,-31.448,46.521,-179.8907,-0.8261,0.0000
C00638=3.695,-27.804,44.865,-179.8395,-1.1765,0.0000
C00639=3.068,-25.489,43.586,175.7793,5.2659,0.0000
C00640=1.615,-24.766,43.062,164.5921,2.6504,0.0000
C00641=0.589,-24.754,43.039,163.4920,-0.4122,0.0000
C00642=0.000,-24.757,43.054,163.5138,-0.0002,0.0000
C00643=0.000,-24.757,43.054,163.5138,-0.0002,0.0000
C00644=-0.589,-24.754,43.039,163.4920,0.4123,0.0000
C00645=-1.615,-24.766,43.062,164.5929,-2.6519,0.0000
C00646=-3.068,-25.489,43.586,175.7798,-5.2656,0.0000
C00647=-3.695,-27.804,44.865,-179.8395,1.1765,0.0000
C00648=-4.151,-31.448,46.521,-179.8907,0.8261,0.0000
C00649=-19.301,-25.172,46.521,179.4931,-0.6614,0.0000
C00650=-17.048,-22.273,44.865,179.2815,-0.9454,0.0000
C00651=-15.854,-20.193,43.586,-179.2457,6.7028,0.0000
C00652=-16.370,-18.654,43.062,170.8582,12.7306,0.0000
C00653=-17.087,-17.920,43.039,167.8734,11.2933,0.0000
C00654=-17.506,-17.506,43.054,168.1802,11.5757,0.0000
C00655=-17.920,-17.087,43.039,168.4559,11.8884,0.0000
C00656=-18.654,-16.370,43.062,167.1106,8.9135,0.0000
C00657=-20.193,-15.854,43.586,173.2972,-0.7493,0.0000
C00658=-22.273,-17.048,44.865,-179.0546,0.7184,0.0000
C00659=-25.172,-19.301,46.521,-179.3386,0.5068,0.0000
C00660=-31.448,-4.151,46.521,179.1739,-0.1093,0.0000
C00661=-27.804,-3.695,44.865,178.8235,-0.1604,0.0000
C00662=-25.489,-3.068,43.586,-174.7199,4.2029,0.0000
C00663=-24.766,-1.615,43.062,-177.2510,15.3911,0.0000
C00664=-24.754,-0.589,43.039,179.5701,16.5075,0.0000
C00665=-24.757,0.000,43.054,179.9998,16.4862,0.0000
C00666=-24.754,0.589,43.039,-179.5700,16.5075,0.0000
C00667=-24.766,1.615,43.062,177.2494,15.3902,0.0000
C00668=-25.489,3.068,43.586,174.7201,4.2024,0.0000
C00669=-27.804,3.695,44.865,-178.8235,-0.1604,0.0000
C00670=-31.448,4.151,46.521,-179.1739,-0.1093,0.0000
C00671=-25.172,19.301,46.521,179.3386,0.5068,0.0000
C00672=-22.273,17.048,44.865,179.0546,0.7184,0.0000
C00673=-20.193,15.854,43.586,-173.2966,-0.7491,0.0000
C00674=-18.654,16.370,43.062,-167.1110,8.9152,0.0000
C00675=-17.920,17.087,43.039,-168.4558,11.8883,0.0000
C00676=-17.506,17.506,43.054,-168.1805,11.5761,0.0000
C00677=-17.087,17.920,43.039,-167.8733,11.2932,0.0000
C00678=-16.370,18.654,43.062,-170.8599,12.7311,0.0000
C00679=-15.854,20.193,43.586,179.2456,6.7022,0.0000
C00680=-17.048,22.273,44.865,-179.2815,-0.9454,0.0000
C00681=-19.301,25.172,46.521,-179.4931,-0.6614,0.0000
C00682=-4.151,31.448,46.521,179.8907,0.8261,0.0000
C00683=-3.695,27.804,44.865,179.8395,1.1765,0.0000
C00684=-3.068,25.489,43.586,-175.7798,-5.2656,0.0000
C00685=-1.615,24.766,43.062,-164.5929,-2.6519,0.0000
C00686=-0.589,24.754,43.039,-163.4920,0.4123,0.0000
C00687=0.000,24.757,43.054,-163.5138,-0.0002,0.0000
C00688=0.000,24.250,45.195,-170.0572,-0.0001,0.0000
C00689=0.543,24.247,45.179,-170.0200,-0.2212,0.0000
C00690=1.537,24.267,45.203,-170.7882,1.6931,0.0000
C00691=2.986,25.071,45.744,-177.8426,2.7768,0.0000
C00692=3.633,27.569,47.051,179.9492,-0.3847,0.0000
C00693=16.925,22.063,47.051,-179.7639,0.3080,0.0000
C00694=15.616,19.839,45.744,179.5599,-3.4882,0.0000
C00695=16.072,18.246,45.203,-174.6583,-7.7031,0.0000
C00696=16.761,17.529,45.179,-172.7509,-6.8814,0.0000
C00697=17.148,17.148,45.195,-172.9339,-7.0129,0.0000
C00698=17.529,16.762,45.179,-173.0637,-7.1966,0.0000
C00699=18.246,16.072,45.203,-172.2635,-5.2923,0.0000
C00700=19.839,15.616,45.744,-176.5120,0.4394,0.0000
C00701=22.063,16.925,47.051,179.6920,-0.2361,0.0000
C00702=27.569,3.633,47.051,-179.6153,0.0508,0.0000
C00703=25.071,2.986,45.744,177.2213,-2.1549,0.0000
C00704=24.267,1.537,45.203,178.2848,-9.2077,0.0000
C00705=24.247,0.543,45.179,-179.7754,-9.9800,0.0000
C00706=24.250,0.000,45.195,-179.9999,-9.9428,0.0000
C00707=24.247,-0.542,45.179,179.7755,-9.9800,0.0000
C00708=24.267,-1.537,45.203,-178.2839,-9.2071,0.0000
C00709=25.071,-2.986,45.744,-177.2215,-2.1546,0.0000
C00710=27.569,-3.633,47.051,179.6153,0.0508,0.0000
C00711=22.063,-16.925,47.051,-179.6920,-0.2361,0.0000
C00712=19.839,-15.616,45.744,176.5117,0.4393,0.0000
C00713=18.246,-16.072,45.203,172.2637,-5.2934,0.0000
C00714=17.529,-16.761,45.179,173.0637,-7.1966,0.0000
C00715=17.148,-17.148,45.195,172.9340,-7.0129,0.0000
C00716=16.762,-17.529,45.179,172.7509,-6.8814,0.0000
C00717=16.072,-18.246,45.203,174.6594,-7.7033,0.0000
C00718=15.616,-19.839,45.744,-179.5598,-3.4879,0.0000
C00719=16.925,-22.063,47.051,179.7639,0.3080,0.0000
C00720=3.633,-27.569,47.051,-179.9492,-0.3847,0.0000
C00721=2.986,-25.071,45.744,177.8426,2.7768,0.0000
C00722=1.537,-24.267,45.203,170.7882,1.6931,0.0000
C00723=0.543,-24.247,45.179,170.0200,-0.2212,0.0000
C00724=0.000,-24.250,45.195,170.0572,-0.0001,0.0000
C00725=0.000,-24.250,45.195,170.0572,-0.0001,0.0000
C00726=-0.542,-24.247,45.179,170.0200,0.2211,0.0000
C00727=-1.537,-24.267,45.203,170.7888,-1.6940,0.0000
C00728=-2.986,-25.071,45.744,177.8429,-2.7766,0.0000
C00729=-3.633,-27.569,47.051,-179.9492,0.3847,0.0000
C00730=-16.925,-22.063,47.051,179.7639,-0.3080,0.0000
C00731=-15.616,-19.839,45.744,-179.5599,3.4882,0.0000
C00732=-16.072,-18.246,45.203,174.6583,7.7031,0.0000
C00733=-16.761,-17.529,45.179,172.7509,6.8814,0.0000
C00734=-17.148,-17.148,45.195,172.9339,7.0129,0.0000
C00735=-17.529,-16.762,45.179,173.0637,7.1966,0.0000
C00736=-18.246,-16.072,45.203,172.2635,5.2923,0.0000
C00737=-19.839,-15.616,45.744,176.5120,-0.4394,0.0000
C00738=-22.063,-16.925,47.051,-179.6920,0.2361,0.0000
C00739=-27.569,-3.633,47.051,179.6153,-0.0508,0.0000
C00740=-25.071,-2.986,45.744,-177.2213,2.1549,0.0000
C00741=-24.267,-1.537,45.203,-178.2848,9.2077,0.0000
C00742=-24.247,-0.543,45.179,179.7754,9.9800,0.0000
C00743=-24.250,0.000,45.195,179.9999,9.9428,0.0000
C00744=-24.247,0.542,45.179,-179.7755,9.9800,0.0000
C00745=-24.267,1.537,45.203,178.2839,9.2071,0.0000
C00746=-25.071,2.986,45.744,177.2215,2.1546,0.0000
C00747=-27.569,3.633,47.051,-179.6153,-0.0508,0.0000
C00748=-22.063,16.925,47.051,179.6920,0.2361,0.0000
C00749=-19.839,15.616,45.744,-176.5117,-0.4393,0.0000
C00750=-18.246,16.072,45.203,-172.2637,5.2934,0.0000
C00751=-17.529,16.761,45.179,-173.0637,7.1966,0.0000
C00752=-17.148,17.148,45.195,-172.9340,7.0129,0.0000
C00753=-16.762,17.529,45.179,-172.7509,6.8814,0.0000
C00754=-16.072,18.246,45.203,-174.6594,7.7033,0.0000
C00755=-15.616,19.839,45.744,179.5598,3.4879,0.0000
C00756=-16.925,22.063,47.051,-179.7639,-0.3080,0.0000
C00757=-3.633,27.569,47.051,179.9492,0.3847,0.0000
C00758=-2.986,25.071,45.744,-177.8429,-2.7766,0.0000
C00759=-1.537,24.267,45.203,-170.7888,-1.6940,0.0000
C00760=-0.542,24.247,45.179,-170.0200,0.2211,0.0000
C00761=0.000,24.250,45.195,-170.0572,-0.0001,0.0000
C00762=0.000,24.012,47.382,-177.6951,-0.0000,0.0000
C00763=0.521,24.008,47.366,-177.6395,-0.0488,0.0000
C00764=1.501,24.033,47.390,-177.8943,0.3992,0.0000
C00765=2.955,24.917,47.939,-179.9400,0.0782,0.0000
C00766=15.529,19.709,47.939,179.9872,-0.0977,0.0000
C00767=15.933,18.055,47.390,-178.7930,-1.7711,0.0000
C00768=16.608,17.344,47.366,-178.2959,-1.6344,0.0000
C00769=16.979,16.979,47.382,-178.3698,-1.6296,0.0000
C00770=17.344,16.608,47.366,-178.3649,-1.7034,0.0000
C00771=18.055,15.933,47.390,-178.2286,-1.2060,0.0000
C00772=19.709,15.529,47.939,-179.9024,0.0128,0.0000
C00773=24.917,2.955,47.939,179.9218,-0.0600,0.0000
C00774=24.033,1.501,47.390,179.6005,-2.1056,0.0000
C00775=24.008,0.521,47.366,-179.9512,-2.3605,0.0000
C00776=24.012,0.000,47.382,-180.0000,-2.3049,0.0000
C00777=24.008,-0.521,47.366,179.9512,-2.3605,0.0000
C00778=24.033,-1.501,47.390,-179.6004,-2.1053,0.0000
C00779=24.917,-2.955,47.939,-179.9219,-0.0600,0.0000
C00780=19.709,-15.529,47.939,179.9023,0.0128,0.0000
C00781=18.055,-15.933,47.390,178.2285,-1.2064,0.0000
C00782=17.344,-16.608,47.366,178.3649,-1.7034,0.0000
C00783=16.979,-16.979,47.382,178.3698,-1.6296,0.0000
C00784=16.608,-17.344,47.366,178.2959,-1.6344,0.0000
C00785=15.933,-18.055,47.390,178.7934,-1.7710,0.0000
C00786=15.529,-19.709,47.939,-179.9872,-0.0976,0.0000
C00787=2.955,-24.917,47.939,179.9400,0.0782,0.0000
C00788=1.501,-24.033,47.390,177.8943,0.3992,0.0000
C00789=0.521,-24.008,47.366,177.6395,-0.0488,0.0000
C00790=0.000,-24.012,47.382,177.6951,-0.0000,0.0000
C00791=0.000,-24.012,47.382,177.6951,-0.0000,0.0000
C00792=-0.521,-24.008,47.366,177.6395,0.0488,0.0000
C00793=-1.501,-24.033,47.390,177.8946,-0.3994,0.0000
C00794=-2.955,-24.917,47.939,179.9400,-0.0781,0.0000
C00795=-15.529,-19.709,47.939,-179.9872,0.0977,0.0000
C00796=-15.933,-18.055,47.390,178.7930,1.7711,0.0000
C00797=-16.608,-17.344,47.366,178.2959,1.6344,0.0000
C00798=-16.979,-16.979,47.382,178.3698,1.6296,0.0000
C00799=-17.344,-16.608,47.366,178.3649,1.7034,0.0000
C00800=-18.055,-15.933,47.390,178.2286,1.2060,0.0000
C00801=-19.709,-15.529,47.939,179.9024,-0.0128,0.0000
C00802=-24.917,-2.955,47.939,-179.9218,0.0600,0.0000
C00803=-24.033,-1.501,47.390,-179.6005,2.1056,0.0000
C00804=-24.008,-0.521,47.366,179.9512,2.3605,0.0000
C00805=-24.012,0.000,47.382,180.0000,2.3049,0.0000
C00806=-24.008,0.521,47.366,-179.9512,2.3605,0.0000
C00807=-24.033,1.501,47.390,179.6004,2.1053,0.0000
C00808=-24.917,2.955,47.939,179.9219,0.0600,0.0000
C00809=-19.709,15.529,47.939,-179.9023,-0.0128,0.0000
C00810=-18.055,15.933,47.390,-178.2285,1.2064,0.0000
C00811=-17.344,16.608,47.366,-178.3649,1.7034,0.0000
C00812=-16.979,16.979,47.382,-178.3698,1.6296,0.0000
C00813=-16.608,17.344,47.366,-178.2959,1.6344,0.0000
C00814=-15.933,18.055,47.390,-178.7934,1.7710,0.0000
C00815=-15.529,19.709,47.939,179.9872,0.0976,0.0000
C00816=-2.955,24.917,47.939,-179.9400,-0.0781,0.0000
C00817=-1.501,24.033,47.390,-177.8946,-0.3994,0.0000
C00818=-0.521,24.008,47.366,-177.6395,0.0488,0.0000
C00819=0.000,24.012,47.382,-177.6951,-0.0000,0.0000
//INST
///DATE 2021/02/10 13:51
///COMM
///ATTR SC,RW,RJ
////FRAME USER 2
///GROUP1 RB1
NOP
MOVL C00000
MOVL C00001
MOVL C00002
MOVL C00003
MOVL C00004
MOVL C00005
MOVL C00006
MOVL C00007
MOVL C00008
MOVL C00009
MOVL C00010
MOVL C00011
MOVL C00012
MOVL C00013
MOVL C00014
MOVL C00015
MOVL C00016
MOVL C00017
MOVL C00018
MOVL C00019
MOVL C00020
MOVL C00021
MOVL C00022
MOVL C00023
MOVL C00024
MOVL C00025
MOVL C00026
MOVL C00027
MOVL C00028
MOVL C00029
MOVL C00030
MOVL C00031
MOVL C00032
MOVL C00033
MOVL C00034
MOVL C00035
MOVL C00036
MOVL C00037
MOVL C00038
MOVL C00039
MOVL C00040
MOVL C00041
MOVL C00042
MOVL C00043
MOVL C00044
MOVL C00045
MOVL C00046
MOVL C00047
MOVL C00048
MOVL C00049
MOVL C00050
MOVL C00051
MOVL C00052
MOVL C00053
MOVL C00054
MOVL C00055
MOVL C00056
MOVL C00057
MOVL C00058
MOVL C00059
MOVL C00060
MOVL C00061
MOVL C00062
MOVL C00063
MOVL C00064
MOVL C00065
MOVL C00066
MOVL C00067
MOVL C00068
MOVL C00069
MOVL C00070
MOVL C00071
MOVL C00072
MOVL C00073
MOVL C00074
MOVL C00075
MOVL C00076
MOVL C00077
MOVL C00078
MOVL C00079
MOVL C00080
MOVL C00081
MOVL C00082
MOVL C00083
MOVL C00084
MOVL C00085
MOVL C00086
MOVL C00087
MOVL C00088
MOVL C00089
MOVL C00090
MOVL C00091
MOVL C00092
MOVL C00093
MOVL C00094
MOVL C00095
MOVL C00096
MOVL C00097
MOVL C00098
MOVL C00099
MOVL C00100
MOVL C00101
MOVL C00102
MOVL C00103
MOVL C00104
MOVL C00105
MOVL C00106
MOVL C00107
MOVL C00108
MOVL C00109
MOVL C00110
MOVL C00111
MOVL C00112
MOVL C00113
MOVL C00114
MOVL C00115
MOVL C00116
MOVL C00117
MOVL C00118
MOVL C00119
MOVL C00120
MOVL C00121
MOVL C00122
MOVL C00123
MOVL C00124
MOVL C00125
MOVL C00126
MOVL C00127
MOVL C00128
MOVL C00129
MOVL C00130
MOVL C00131
MOVL C00132
MOVL C00133
MOVL C00134
MOVL C00135
MOVL C00136
MOVL C00137
MOVL C00138
MOVL C00139
MOVL C00140
MOVL C00141
MOVL C00142
MOVL C00143
MOVL C00144
MOVL C00145
MOVL C00146
MOVL C00147
MOVL C00148
MOVL C00149
MOVL C00150
MOVL C00151
MOVL C00152
MOVL C00153
MOVL C00154
MOVL C00155
MOVL C00156
MOVL C00157
MOVL C00158
MOVL C00159
MOVL C00160
MOVL C00161
MOVL C00162
MOVL C00163
MOVL C00164
MOVL C00165
MOVL C00166
MOVL C00167
MOVL C00168
MOVL C00169
MOVL C00170
MOVL C00171
MOVL C00172
MOVL C00173
MOVL C00174
MOVL C00175
MOVL C00176
MOVL C00177
MOVL C00178
MOVL C00179
MOVL C00180
MOVL C00181
MOVL C00182
MOVL C00183
MOVL C00184
MOVL C00185
MOVL C00186
MOVL C00187
MOVL C00188
MOVL C00189
MOVL C00190
MOVL C00191
MOVL C00192
MOVL C00193
MOVL C00194
MOVL C00195
MOVL C00196
MOVL C00197
MOVL C00198
MOVL C00199
MOVL C00200
MOVL C00201
MOVL C00202
MOVL C00203
MOVL C00204
MOVL C00205
MOVL C00206
MOVL C00207
MOVL C00208
MOVL C00209
MOVL C00210
MOVL C00211
MOVL C00212
MOVL C00213
MOVL C00214
MOVL C00215
MOVL C00216
MOVL C00217
MOVL C00218
MOVL C00219
MOVL C00220
MOVL C00221
MOVL C00222
MOVL C00223
MOVL C00224
MOVL C00225
MOVL C00226
MOVL C00227
MOVL C00228
MOVL C00229
MOVL C00230
MOVL C00231
MOVL C00232
MOVL C00233
MOVL C00234
MOVL C00235
MOVL C00236
MOVL C00237
MOVL C00238
MOVL C00239
MOVL C00240
MOVL C00241
MOVL C00242
MOVL C00243
MOVL C00244
MOVL C00245
MOVL C00246
MOVL C00247
MOVL C00248
MOVL C00249
MOVL C00250
MOVL C00251
MOVL C00252
MOVL C00253
MOVL C00254
MOVL C00255
MOVL C00256
MOVL C00257
MOVL C00258
MOVL C00259
MOVL C00260
MOVL C00261
MOVL C00262
MOVL C00263
MOVL C00264
MOVL C00265
MOVL C00266
MOVL C00267
MOVL C00268
MOVL C00269
MOVL C00270
MOVL C00271
MOVL C00272
MOVL C00273
MOVL C00274
MOVL C00275
MOVL C00276
MOVL C00277
MOVL C00278
MOVL C00279
MOVL C00280
MOVL C00281
MOVL C00282
MOVL C00283
MOVL C00284
MOVL C00285
MOVL C00286
MOVL C00287
MOVL C00288
MOVL C00289
MOVL C00290
MOVL C00291
MOVL C00292
MOVL C00293
MOVL C00294
MOVL C00295
MOVL C00296
MOVL C00297
MOVL C00298
MOVL C00299
MOVL C00300
MOVL C00301
MOVL C00302
MOVL C00303
MOVL C00304
MOVL C00305
MOVL C00306
MOVL C00307
MOVL C00308
MOVL C00309
MOVL C00310
MOVL C00311
MOVL C00312
MOVL C00313
MOVL C00314
MOVL C00315
MOVL C00316
MOVL C00317
MOVL C00318
MOVL C00319
MOVL C00320
MOVL C00321
MOVL C00322
MOVL C00323
MOVL C00324
MOVL C00325
MOVL C00326
MOVL C00327
MOVL C00328
MOVL C00329
MOVL C00330
MOVL C00331
MOVL C00332
MOVL C00333
MOVL C00334
MOVL C00335
MOVL C00336
MOVL C00337
MOVL C00338
MOVL C00339
MOVL C00340
MOVL C00341
MOVL C00342
MOVL C00343
MOVL C00344
MOVL C00345
MOVL C00346
MOVL C00347
MOVL C00348
MOVL C00349
MOVL C00350
MOVL C00351
MOVL C00352
MOVL C00353
MOVL C00354
MOVL C00355
MOVL C00356
MOVL C00357
MOVL C00358
MOVL C00359
MOVL C00360
MOVL C00361
MOVL C00362
MOVL C00363
MOVL C00364
MOVL C00365
MOVL C00366
MOVL C00367
MOVL C00368
MOVL C00369
MOVL C00370
MOVL C00371
MOVL C00372
MOVL C00373
MOVL C00374
MOVL C00375
MOVL C00376
MOVL C00377
MOVL C00378
MOVL C00379
MOVL C00380
MOVL C00381
MOVL C00382
MOVL C00383
MOVL C00384
MOVL C00385
MOVL C00386
MOVL C00387
MOVL C00388
MOVL C00389
MOVL C00390
MOVL C00391
MOVL C00392
MOVL C00393
MOVL C00394
MOVL C00395
MOVL C00396
MOVL C00397
MOVL C00398
MOVL C00399
MOVL C00400
MOVL C00401
MOVL C00402
MOVL C00403
MOVL C00404
MOVL C00405
MOVL C00406
MOVL C00407
MOVL C00408
MOVL C00409
MOVL C00410
MOVL C00411
MOVL C00412
MOVL C00413
MOVL C00414
MOVL C00415
MOVL C00416
MOVL C00417
MOVL C00418
MOVL C00419
MOVL C00420
MOVL C00421
MOVL C00422
MOVL C00423
MOVL C00424
MOVL C00425
MOVL C00426
MOVL C00427
MOVL C00428
MOVL C00429
MOVL C00430
MOVL C00431
MOVL C00432
MOVL C00433
MOVL C00434
MOVL C00435
MOVL C00436
MOVL C00437
MOVL C00438
MOVL C00439
MOVL C00440
MOVL C00441
MOVL C00442
MOVL C00443
MOVL C00444
MOVL C00445
MOVL C00446
MOVL C00447
MOVL C00448
MOVL C00449
MOVL C00450
MOVL C00451
MOVL C00452
MOVL C00453
ARCOF
MOVL C00454
ARCON
MOVL C00455
MOVL C00456
MOVL C00457
MOVL C00458
MOVL C00459
MOVL C00460
MOVL C00461
MOVL C00462
MOVL C00463
MOVL C00464
MOVL C00465
MOVL C00466
MOVL C00467
MOVL C00468
MOVL C00469
MOVL C00470
MOVL C00471
MOVL C00472
ARCOF
MOVL C00473
ARCON
MOVL C00474
MOVL C00475
MOVL C00476
MOVL C00477
MOVL C00478
MOVL C00479
MOVL C00480
MOVL C00481
MOVL C00482
MOVL C00483
MOVL C00484
MOVL C00485
MOVL C00486
MOVL C00487
MOVL C00488
MOVL C00489
MOVL C00490
MOVL C00491
ARCOF
MOVL C00492
ARCON
MOVL C00493
MOVL C00494
MOVL C00495
MOVL C00496
MOVL C00497
MOVL C00498
MOVL C00499
MOVL C00500
MOVL C00501
MOVL C00502
MOVL C00503
MOVL C00504
MOVL C00505
MOVL C00506
MOVL C00507
MOVL C00508
MOVL C00509
MOVL C00510
ARCOF
MOVL C00511
ARCON
MOVL C00512
MOVL C00513
MOVL C00514
MOVL C00515
MOVL C00516
MOVL C00517
MOVL C00518
MOVL C00519
MOVL C00520
MOVL C00521
MOVL C00522
MOVL C00523
MOVL C00524
MOVL C00525
MOVL C00526
MOVL C00527
MOVL C00528
MOVL C00529
MOVL C00530
ARCOF
MOVL C00531
ARCON
MOVL C00532
MOVL C00533
MOVL C00534
MOVL C00535
MOVL C00536
MOVL C00537
MOVL C00538
MOVL C00539
MOVL C00540
MOVL C00541
MOVL C00542
MOVL C00543
MOVL C00544
MOVL C00545
MOVL C00546
MOVL C00547
MOVL C00548
MOVL C00549
ARCOF
MOVL C00550
ARCON
MOVL C00551
MOVL C00552
MOVL C00553
MOVL C00554
MOVL C00555
MOVL C00556
MOVL C00557
MOVL C00558
MOVL C00559
MOVL C00560
MOVL C00561
MOVL C00562
MOVL C00563
MOVL C00564
MOVL C00565
MOVL C00566
MOVL C00567
MOVL C00568
ARCOF
MOVL C00569
ARCON
MOVL C00570
MOVL C00571
MOVL C00572
MOVL C00573
MOVL C00574
MOVL C00575
MOVL C00576
MOVL C00577
MOVL C00578
MOVL C00579
MOVL C00580
MOVL C00581
MOVL C00582
MOVL C00583
MOVL C00584
MOVL C00585
MOVL C00586
MOVL C00587
ARCOF
MOVL C00588
ARCON
MOVL C00589
MOVL C00590
MOVL C00591
MOVL C00592
MOVL C00593
MOVL C00594
MOVL C00595
MOVL C00596
MOVL C00597
MOVL C00598
MOVL C00599
MOVL C00600
MOVL C00601
MOVL C00602
MOVL C00603
ARCOF
MOVL C00604
ARCON
MOVL C00605
MOVL C00606
MOVL C00607
MOVL C00608
MOVL C00609
MOVL C00610
MOVL C00611
MOVL C00612
MOVL C00613
MOVL C00614
ARCOF
MOVL C00615
ARCON
MOVL C00616
MOVL C00617
MOVL C00618
MOVL C00619
MOVL C00620
MOVL C00621
MOVL C00622
MOVL C00623
MOVL C00624
MOVL C00625
ARCOF
MOVL C00626
ARCON
MOVL C00627
MOVL C00628
MOVL C00629
MOVL C00630
MOVL C00631
MOVL C00632
MOVL C00633
MOVL C00634
MOVL C00635
MOVL C00636
ARCOF
MOVL C00637
ARCON
MOVL C00638
MOVL C00639
MOVL C00640
MOVL C00641
MOVL C00642
MOVL C00643
MOVL C00644
MOVL C00645
MOVL C00646
MOVL C00647
MOVL C00648
ARCOF
MOVL C00649
ARCON
MOVL C00650
MOVL C00651
MOVL C00652
MOVL C00653
MOVL C00654
MOVL C00655
MOVL C00656
MOVL C00657
MOVL C00658
MOVL C00659
ARCOF
MOVL C00660
ARCON
MOVL C00661
MOVL C00662
MOVL C00663
MOVL C00664
MOVL C00665
MOVL C00666
MOVL C00667
MOVL C00668
MOVL C00669
MOVL C00670
ARCOF
MOVL C00671
ARCON
MOVL C00672
MOVL C00673
MOVL C00674
MOVL C00675
MOVL C00676
MOVL C00677
MOVL C00678
MOVL C00679
MOVL C00680
MOVL C00681
ARCOF
MOVL C00682
ARCON
MOVL C00683
MOVL C00684
MOVL C00685
MOVL C00686
MOVL C00687
MOVL C00688
MOVL C00689
MOVL C00690
MOVL C00691
MOVL C00692
ARCOF
MOVL C00693
ARCON
MOVL C00694
MOVL C00695
MOVL C00696
MOVL C00697
MOVL C00698
MOVL C00699
MOVL C00700
MOVL C00701
ARCOF
MOVL C00702
ARCON
MOVL C00703
MOVL C00704
MOVL C00705
MOVL C00706
MOVL C00707
MOVL C00708
MOVL C00709
MOVL C00710
ARCOF
MOVL C00711
ARCON
MOVL C00712
MOVL C00713
MOVL C00714
MOVL C00715
MOVL C00716
MOVL C00717
MOVL C00718
MOVL C00719
ARCOF
MOVL C00720
ARCON
MOVL C00721
MOVL C00722
MOVL C00723
MOVL C00724
MOVL C00725
MOVL C00726
MOVL C00727
MOVL C00728
MOVL C00729
ARCOF
MOVL C00730
ARCON
MOVL C00731
MOVL C00732
MOVL C00733
MOVL C00734
MOVL C00735
MOVL C00736
MOVL C00737
MOVL C00738
ARCOF
MOVL C00739
ARCON
MOVL C00740
MOVL C00741
MOVL C00742
MOVL C00743
MOVL C00744
MOVL C00745
MOVL C00746
MOVL C00747
ARCOF
MOVL C00748
ARCON
MOVL C00749
MOVL C00750
MOVL C00751
MOVL C00752
MOVL C00753
MOVL C00754
MOVL C00755
MOVL C00756
ARCOF
MOVL C00757
ARCON
MOVL C00758
MOVL C00759
MOVL C00760
MOVL C00761
MOVL C00762
MOVL C00763
MOVL C00764
MOVL C00765
ARCOF
MOVL C00766
ARCON
MOVL C00767
MOVL C00768
MOVL C00769
MOVL C00770
MOVL C00771
MOVL C00772
ARCOF
MOVL C00773
ARCON
MOVL C00774
MOVL C00775
MOVL C00776
MOVL C00777
MOVL C00778
MOVL C00779
ARCOF
MOVL C00780
ARCON
MOVL C00781
MOVL C00782
MOVL C00783
MOVL C00784
MOVL C00785
MOVL C00786
ARCOF
MOVL C00787
ARCON
MOVL C00788
MOVL C00789
MOVL C00790
MOVL C00791
MOVL C00792
MOVL C00793
MOVL C00794
ARCOF
MOVL C00795
ARCON
MOVL C00796
MOVL C00797
MOVL C00798
MOVL C00799
MOVL C00800
MOVL C00801
ARCOF
MOVL C00802
ARCON
MOVL C00803
MOVL C00804
MOVL C00805
MOVL C00806
MOVL C00807
MOVL C00808
ARCOF
MOVL C00809
ARCON
MOVL C00810
MOVL C00811
MOVL C00812
MOVL C00813
MOVL C00814
MOVL C00815
ARCOF
MOVL C00816
ARCON
MOVL C00817
MOVL C00818
MOVL C00819
END
